FUNCTION F_DegToRad : LREAL
VAR_INPUT
	fInputDeg 	: LREAL;
END_VAR
VAR
	fPi 		:LREAL := 3.14159265359;
END_VAR

F_DegToRad := fInputDeg*(fPi/180);

END_FUNCTION

(* stored: Version 1.1.0.1, ProductVersion 3.1.4024.11
   POU F_DegToRad: Id {5200f035-ac36-40d0-a8b8-8b3584a964b4}, SpecialFunc None *)
